(* IEC 61131-3 sources: eCockpitGit/test_project/src/%F%00 Library/%F%Common Functions/%F%Conversion/%F%AnyConversion, 28 files *)

(* ---- %POU%AnyATToSAny.st ---- *)
//This converts a pointer and a type to a sany
// |**Version**|**Author**| **Date** |**Changes**
// | 1         | NSN      | 13-12-19 | Creation
FUNCTION AnyATToSAny : SAny
VAR_INPUT
	pVal		:POINTER TO USysTypes;	//Address of value
	eType		:ESysType;				//Type of value
END_VAR
(*%!%__DELIMITER__%!%*)
AnyATToSAny.eType		:=		eType;
AnyATToSAny.pVal		:=		pVal;

(* ---- %POU%AnyToSAny.st ---- *)
//This function converts any variable to a sany
// |**Version**|**Author**| **Date** |**Changes**
// | 1         | NSN      | 13-12-19 | Creation
FUNCTION AnyToSAny : SAny
VAR_INPUT
	aAnyIn	:ANY;
END_VAR
(*%!%__DELIMITER__%!%*)
AnyToSAny.eType		:=		TO_BYTE(aAnyIn.TypeClass);
AnyToSAny.pVal		:=		aAnyIn.pValue;

(* ---- %POU%BitToSVar.st ---- *)
//This function get the bit value from a variable
// |**Version**|**Author**| **Date** |**Changes**
// | 1         | NSN      | 11-01-19 | Creation
FUNCTION BitToSVar : BOOL
VAR_INPUT
	xBit	:BOOL;		//Bool to set
	sVar	:SVar;		//Variable to get bit value from
END_VAR
(*%!%__DELIMITER__%!%*)
CASE sVar.bOffset OF
	1..8:	sVar.sAny.pVal^.bBYTE	:=		(sVar.sAny.pVal^.bBYTE AND NOT(SHL(TO_BYTE(1),sVar.bOffset-1))) OR (SHL(TO_BYTE(xBit),sVar.bOffset-1));
	9..16:	sVar.sAny.pVal^.bWORD	:=		(sVar.sAny.pVal^.bWORD AND NOT(SHL(TO_WORD(1),sVar.bOffset-1))) OR (SHL(TO_WORD(xBit),sVar.bOffset-1));
	17..32:	sVar.sAny.pVal^.bDWORD	:=		(sVar.sAny.pVal^.bDWORD AND NOT(SHL(TO_DWORD(1),sVar.bOffset-1))) OR (SHL(TO_DWORD(xBit),sVar.bOffset-1));
END_CASE

(* ---- %POU%BOOLToSAny.st ---- *)
//This function converts a dint to any variable
// |**Version**|**Author**| **Date** |**Changes**
// | 1         | NSN      | 23-07-18 | Creation
FUNCTION BOOLToSAny : BOOL
VAR_INPUT
	in			:BOOL;		//Input variable
	sOut		:SAny;		//Variable information
END_VAR
(*%!%__DELIMITER__%!%*)
CASE sOut.eType OF
	ESysType.tBOOL:		//Bool conversion
		sOut.pVal^.bBOOL		:=		in;
	ESysType.tBYTE:
		sOut.pVal^.bBYTE		:=		TO_BYTE(in);
	ESysType.tWORD:
		sOut.pVal^.bWORD		:=		TO_WORD(in);
	ESysType.tDWORD:
		sOut.pVal^.bDWORD		:=		TO_DWORD(in);
	ESysType.tLWORD:
		sOut.pVal^.bLWORD		:=		TO_LWORD(in);
	ESysType.tSINT:
		sOut.pVal^.bSINT		:=		TO_SINT(in);
	ESysType.tINT:
		sOut.pVal^.bINT			:=		TO_INT(in);
	ESysType.tDINT:
		sOut.pVal^.bDINT		:=		TO_DINT(in);
	ESysType.tLINT:
		sOut.pVal^.bLINT		:=		TO_LINT(in);
	ESysType.tUSINT:
		sOut.pVal^.bUSINT		:=		TO_USINT(in);
	ESysType.tUINT:
		sOut.pVal^.bUINT		:=		TO_UINT(in);
	ESysType.tUDINT:
		sOut.pVal^.bUDINT		:=		TO_UDINT(in);
	ESysType.tULINT:
		sOut.pVal^.bULINT		:=		TO_ULINT(in);
	ESysType.tREAL:
		sOut.pVal^.bREAL		:=		TO_REAL(in);
	ESysType.tLREAL:
		sOut.pVal^.bLREAL		:=		TO_LREAL(in);
	ESysType.tSTRING:
		sOut.pVal^.bSTRING		:=		TO_STRING(in);
	ESysType.tTIME:
		sOut.pVal^.bTIME		:=		TO_TIME(in);
	ESysType.tDATE:
		sOut.pVal^.bDATE		:=		TO_DATE(in);
	ESysType.tDT:
		sOut.pVal^.bDT			:=		TO_DT(in);
	ESysType.tTOD:
		sOut.pVal^.bTOD			:=		TO_TOD(in);
	ESysType.tLTIME:
		sOut.pVal^.bLTIME		:=		TO_LTIME(in);
ELSE
	RETURN;
END_CASE

(* ---- %POU%DINTToSAny.st ---- *)
//This function converts a dint to any variable
// |**Version**|**Author**| **Date** |**Changes**
// | 1         | NSN      | 23-07-18 | Creation
FUNCTION DINTToSAny : BOOL
VAR_INPUT
	in			:DINT;		//Input variable
	sOut		:SAny;		//Variable information
END_VAR
(*%!%__DELIMITER__%!%*)
CASE sOut.eType OF
	ESysType.tBOOL:		//Bool conversion
		sOut.pVal^.bBOOL		:=		TO_BOOL(in);
	ESysType.tBYTE:
		sOut.pVal^.bBYTE		:=		TO_BYTE(in);
	ESysType.tWORD:
		sOut.pVal^.bWORD		:=		TO_WORD(in);
	ESysType.tDWORD:
		sOut.pVal^.bDWORD		:=		TO_DWORD(in);
	ESysType.tLWORD:
		sOut.pVal^.bLWORD		:=		TO_LWORD(in);
	ESysType.tSINT:
		sOut.pVal^.bSINT		:=		TO_SINT(in);
	ESysType.tINT:
		sOut.pVal^.bINT			:=		TO_INT(in);
	ESysType.tDINT:
		sOut.pVal^.bDINT		:=		in;
	ESysType.tLINT:
		sOut.pVal^.bLINT		:=		in;
	ESysType.tUSINT:
		sOut.pVal^.bUSINT		:=		TO_USINT(in);
	ESysType.tUINT:
		sOut.pVal^.bUINT		:=		TO_UINT(in);
	ESysType.tUDINT:
		sOut.pVal^.bUDINT		:=		TO_UDINT(in);
	ESysType.tULINT:
		sOut.pVal^.bULINT		:=		TO_ULINT(in);
	ESysType.tREAL:
		sOut.pVal^.bREAL		:=		TO_REAL(in);
	ESysType.tLREAL:
		sOut.pVal^.bLREAL		:=		TO_LREAL(in);
	ESysType.tSTRING:
		sOut.pVal^.bSTRING		:=		TO_STRING(in);
	ESysType.tTIME:
		sOut.pVal^.bTIME		:=		TO_TIME(in);
	ESysType.tDATE:
		sOut.pVal^.bDATE		:=		TO_DATE(in);
	ESysType.tDT:
		sOut.pVal^.bDT			:=		TO_DT(in);
	ESysType.tTOD:
		sOut.pVal^.bTOD			:=		TO_TOD(in);
	ESysType.tLTIME:
		sOut.pVal^.bLTIME		:=		TO_LTIME(in);
ELSE
	RETURN;
END_CASE

(* ---- %POU%SAnyToBOOL.st ---- *)
//This function converts any type from the type and address to a real
// |**Version**|**Author**| **Date** |**Changes**
// | 1         | NSN      | 23-07-18 | Creation
FUNCTION SAnyToBOOL : BOOL
VAR_INPUT
	sAny		:SAny;		//Variable information
END_VAR
(*%!%__DELIMITER__%!%*)
CASE sAny.eType OF
	ESysType.tBOOL:		//Bool conversion
		SAnyToBOOL			:=		sAny.pVal^.bBOOL;
	ESysType.tBYTE:
		SAnyToBOOL			:=		TO_BOOL(sAny.pVal^.bBYTE);
	ESysType.tWORD:
		SAnyToBOOL			:=		TO_BOOL(sAny.pVal^.bWORD);
	ESysType.tDWORD:
		SAnyToBOOL			:=		TO_BOOL(sAny.pVal^.bDWORD);
	ESysType.tLWORD:
		SAnyToBOOL			:=		TO_BOOL(sAny.pVal^.bLWORD);
	ESysType.tSINT:
		SAnyToBOOL			:=		TO_BOOL(sAny.pVal^.bSINT);
	ESysType.tINT:
		SAnyToBOOL			:=		TO_BOOL(sAny.pVal^.bINT);
	ESysType.tDINT:
		SAnyToBOOL			:=		TO_BOOL(sAny.pVal^.bDINT);
	ESysType.tLINT:
		SAnyToBOOL			:=		TO_BOOL(sAny.pVal^.bLINT);
	ESysType.tUSINT:
		SAnyToBOOL			:=		TO_BOOL(sAny.pVal^.bUSINT);
	ESysType.tUINT:
		SAnyToBOOL			:=		TO_BOOL(sAny.pVal^.bUINT);
	ESysType.tUDINT:
		SAnyToBOOL			:=		TO_BOOL(sAny.pVal^.bUDINT);
	ESysType.tULINT:
		SAnyToBOOL			:=		TO_BOOL(sAny.pVal^.bULINT);
	ESysType.tREAL:
		SAnyToBOOL			:=		TO_BOOL(sAny.pVal^.bREAL);
	ESysType.tLREAL:
		SAnyToBOOL			:=		TO_BOOL(sAny.pVal^.bLREAL);
	ESysType.tSTRING:
		SAnyToBOOL			:=		TO_BOOL(sAny.pVal^.bSTRING);
	ESysType.tTIME:
		SAnyToBOOL			:=		TO_BOOL(sAny.pVal^.bTIME);
	ESysType.tDATE:
		SAnyToBOOL			:=		TO_BOOL(sAny.pVal^.bDATE);
	ESysType.tDT:
		SAnyToBOOL			:=		TO_BOOL(sAny.pVal^.bDT);
	ESysType.tTOD:
		SAnyToBOOL			:=		TO_BOOL(sAny.pVal^.bTOD);
	ESysType.tLTIME:
		SAnyToBOOL			:=		TO_BOOL(sAny.pVal^.bLTIME);
ELSE
	RETURN;
END_CASE

(* ---- %POU%SAnyToBYTE.st ---- *)
//This function converts any type from the type and address to a real
// |**Version**|**Author**| **Date** |**Changes**
// | 1         | NSN      | 23-07-18 | Creation
FUNCTION SAnyToBYTE : BYTE
VAR_INPUT
	sAny		:SAny;		//Variable information
END_VAR
(*%!%__DELIMITER__%!%*)
CASE sAny.eType OF
	ESysType.tBOOL:		//Bool conversion
		SAnyToBYTE			:=		TO_BYTE(sAny.pVal^.bBOOL);
	ESysType.tBYTE:
		SAnyToBYTE			:=		sAny.pVal^.bBYTE;
	ESysType.tWORD:
		SAnyToBYTE			:=		TO_BYTE(sAny.pVal^.bWORD);
	ESysType.tDWORD:
		SAnyToBYTE			:=		TO_BYTE(sAny.pVal^.bDWORD);
	ESysType.tLWORD:
		SAnyToBYTE			:=		TO_BYTE(sAny.pVal^.bLWORD);
	ESysType.tSINT:
		SAnyToBYTE			:=		TO_BYTE(sAny.pVal^.bSINT);
	ESysType.tINT:
		SAnyToBYTE			:=		TO_BYTE(sAny.pVal^.bINT);
	ESysType.tDINT:
		SAnyToBYTE			:=		TO_BYTE(sAny.pVal^.bDINT);
	ESysType.tLINT:
		SAnyToBYTE			:=		TO_BYTE(sAny.pVal^.bLINT);
	ESysType.tUSINT:
		SAnyToBYTE			:=		TO_BYTE(sAny.pVal^.bUSINT);
	ESysType.tUINT:
		SAnyToBYTE			:=		TO_BYTE(sAny.pVal^.bUINT);
	ESysType.tUDINT:
		SAnyToBYTE			:=		TO_BYTE(sAny.pVal^.bUDINT);
	ESysType.tULINT:
		SAnyToBYTE			:=		TO_BYTE(sAny.pVal^.bULINT);
	ESysType.tREAL:
		SAnyToBYTE			:=		TO_BYTE(sAny.pVal^.bREAL);
	ESysType.tLREAL:
		SAnyToBYTE			:=		TO_BYTE(sAny.pVal^.bLREAL);
	ESysType.tSTRING:
		SAnyToBYTE			:=		TO_BYTE(sAny.pVal^.bSTRING);
	ESysType.tTIME:
		SAnyToBYTE			:=		TO_BYTE(sAny.pVal^.bTIME);
	ESysType.tDATE:
		SAnyToBYTE			:=		TO_BYTE(sAny.pVal^.bDATE);
	ESysType.tDT:
		SAnyToBYTE			:=		TO_BYTE(sAny.pVal^.bDT);
	ESysType.tTOD:
		SAnyToBYTE			:=		TO_BYTE(sAny.pVal^.bTOD);
	ESysType.tLTIME:
		SAnyToBYTE			:=		TO_BYTE(sAny.pVal^.bLTIME);
ELSE
	RETURN;
END_CASE

(* ---- %POU%SAnyToDATE.st ---- *)
//This function converts any type from the type and address to a real
// |**Version**|**Author**| **Date** |**Changes**
// | 1         | NSN      | 23-07-18 | Creation
FUNCTION SAnyToDATE : DATE
VAR_INPUT
	sAny		:SAny;		//Variable information
END_VAR
(*%!%__DELIMITER__%!%*)
CASE sAny.eType OF
	ESysType.tBOOL:		//Bool conversion
		SAnyToDATE			:=		TO_DATE(sAny.pVal^.bBOOL);
	ESysType.tBYTE:
		SAnyToDATE			:=		TO_DATE(sAny.pVal^.bBYTE);
	ESysType.tWORD:
		SAnyToDATE			:=		TO_DATE(sAny.pVal^.bWORD);
	ESysType.tDWORD:
		SAnyToDATE			:=		TO_DATE(sAny.pVal^.bDWORD);
	ESysType.tLWORD:
		SAnyToDATE			:=		TO_DATE(sAny.pVal^.bLWORD);
	ESysType.tSINT:
		SAnyToDATE			:=		TO_DATE(sAny.pVal^.bSINT);
	ESysType.tINT:
		SAnyToDATE			:=		TO_DATE(sAny.pVal^.bINT);
	ESysType.tDINT:
		SAnyToDATE			:=		TO_DATE(sAny.pVal^.bDINT);
	ESysType.tLINT:
		SAnyToDATE			:=		TO_DATE(sAny.pVal^.bLINT);
	ESysType.tUSINT:
		SAnyToDATE			:=		TO_DATE(sAny.pVal^.bUSINT);
	ESysType.tUINT:
		SAnyToDATE			:=		TO_DATE(sAny.pVal^.bUINT);
	ESysType.tUDINT:
		SAnyToDATE			:=		TO_DATE(sAny.pVal^.bUDINT);
	ESysType.tULINT:
		SAnyToDATE			:=		TO_DATE(sAny.pVal^.bULINT);
	ESysType.tREAL:
		SAnyToDATE			:=		TO_DATE(sAny.pVal^.bREAL);
	ESysType.tLREAL:
		SAnyToDATE			:=		TO_DATE(sAny.pVal^.bLREAL);
	ESysType.tSTRING:
		SAnyToDATE			:=		TO_DATE(sAny.pVal^.bSTRING);
	ESysType.tTIME:
		SAnyToDATE			:=		TO_DATE(sAny.pVal^.bTIME);
	ESysType.tDATE:
		SAnyToDATE			:=		sAny.pVal^.bDATE;
	ESysType.tDT:
		SAnyToDATE			:=		TO_DATE(sAny.pVal^.bDT);
	ESysType.tTOD:
		SAnyToDATE			:=		TO_DATE(sAny.pVal^.bTOD);
	ESysType.tLTIME:
		SAnyToDATE			:=		TO_DATE(sAny.pVal^.bLTIME);
ELSE
	RETURN;
END_CASE

(* ---- %POU%SAnyToDINT.st ---- *)
//This function converts any type from the type and address to a real
// |**Version**|**Author**| **Date** |**Changes**
// | 1         | NSN      | 23-07-18 | Creation
FUNCTION SAnyToDINT : DINT
VAR_INPUT
	sAny		:SAny;		//Variable information
END_VAR
(*%!%__DELIMITER__%!%*)
CASE sAny.eType OF
	ESysType.tBOOL:		//Bool conversion
		SAnyToDINT			:=		TO_DINT(sAny.pVal^.bBOOL);
	ESysType.tBYTE:
		SAnyToDINT			:=		sAny.pVal^.bBYTE;
	ESysType.tWORD:
		SAnyToDINT			:=		sAny.pVal^.bWORD;
	ESysType.tDWORD:
		SAnyToDINT			:=		TO_DINT(sAny.pVal^.bDWORD);
	ESysType.tLWORD:
		SAnyToDINT			:=		TO_DINT(sAny.pVal^.bLWORD);
	ESysType.tSINT:
		SAnyToDINT			:=		sAny.pVal^.bSINT;
	ESysType.tINT:
		SAnyToDINT			:=		sAny.pVal^.bINT;
	ESysType.tDINT:
		SAnyToDINT			:=		sAny.pVal^.bDINT;
	ESysType.tLINT:
		SAnyToDINT			:=		TO_DINT(sAny.pVal^.bLINT);
	ESysType.tUSINT:
		SAnyToDINT			:=		sAny.pVal^.bUSINT;
	ESysType.tUINT:
		SAnyToDINT			:=		sAny.pVal^.bUINT;
	ESysType.tUDINT:
		SAnyToDINT			:=		TO_DINT(sAny.pVal^.bUDINT);
	ESysType.tULINT:
		SAnyToDINT			:=		TO_DINT(sAny.pVal^.bULINT);
	ESysType.tREAL:
		SAnyToDINT			:=		TO_DINT(sAny.pVal^.bREAL);
	ESysType.tLREAL:
		SAnyToDINT			:=		TO_DINT(sAny.pVal^.bLREAL);
	ESysType.tSTRING:
		SAnyToDINT			:=		TO_DINT(sAny.pVal^.bSTRING);
	ESysType.tTIME:
		SAnyToDINT			:=		TO_DINT(sAny.pVal^.bTIME);
	ESysType.tDATE:
		SAnyToDINT			:=		TO_DINT(sAny.pVal^.bDATE);
	ESysType.tDT:
		SAnyToDINT			:=		TO_DINT(sAny.pVal^.bDT);
	ESysType.tTOD:
		SAnyToDINT			:=		TO_DINT(sAny.pVal^.bTOD);
	ESysType.tLTIME:
		SAnyToDINT			:=		TO_DINT(sAny.pVal^.bLTIME);
ELSE
	RETURN;
END_CASE

(* ---- %POU%SAnyToDT.st ---- *)
//This function converts any type from the type and address to a real
// |**Version**|**Author**| **Date** |**Changes**
// | 1         | NSN      | 23-07-18 | Creation
FUNCTION SAnyToDT : DT
VAR_INPUT
	sAny		:SAny;		//Variable information
END_VAR
(*%!%__DELIMITER__%!%*)
CASE sAny.eType OF
	ESysType.tBOOL:		//Bool conversion
		SAnyToDT			:=		TO_DT(sAny.pVal^.bBOOL);
	ESysType.tBYTE:
		SAnyToDT			:=		TO_DT(sAny.pVal^.bBYTE);
	ESysType.tWORD:
		SAnyToDT			:=		TO_DT(sAny.pVal^.bWORD);
	ESysType.tDWORD:
		SAnyToDT			:=		TO_DT(sAny.pVal^.bDWORD);
	ESysType.tLWORD:
		SAnyToDT			:=		TO_DT(sAny.pVal^.bLWORD);
	ESysType.tSINT:
		SAnyToDT			:=		TO_DT(sAny.pVal^.bSINT);
	ESysType.tINT:
		SAnyToDT			:=		TO_DT(sAny.pVal^.bINT);
	ESysType.tDINT:
		SAnyToDT			:=		TO_DT(sAny.pVal^.bDINT);
	ESysType.tLINT:
		SAnyToDT			:=		TO_DT(sAny.pVal^.bLINT);
	ESysType.tUSINT:
		SAnyToDT			:=		TO_DT(sAny.pVal^.bUSINT);
	ESysType.tUINT:
		SAnyToDT			:=		TO_DT(sAny.pVal^.bUINT);
	ESysType.tUDINT:
		SAnyToDT			:=		TO_DT(sAny.pVal^.bUDINT);
	ESysType.tULINT:
		SAnyToDT			:=		TO_DT(sAny.pVal^.bULINT);
	ESysType.tREAL:
		SAnyToDT			:=		TO_DT(sAny.pVal^.bREAL);
	ESysType.tLREAL:
		SAnyToDT			:=		TO_DT(sAny.pVal^.bLREAL);
	ESysType.tSTRING:
		SAnyToDT			:=		TO_DT(sAny.pVal^.bSTRING);
	ESysType.tTIME:
		SAnyToDT			:=		TO_DT(sAny.pVal^.bTIME);
	ESysType.tDATE:
		SAnyToDT			:=		TO_DT(sAny.pVal^.bDATE);
	ESysType.tDT:
		SAnyToDT			:=		sAny.pVal^.bDT;
	ESysType.tTOD:
		SAnyToDT			:=		TO_DT(sAny.pVal^.bTOD);
	ESysType.tLTIME:
		SAnyToDT			:=		TO_DT(sAny.pVal^.bLTIME);
ELSE
	RETURN;
END_CASE

(* ---- %POU%SAnyToDWORD.st ---- *)
//This function converts any type from the type and address to a real
// |**Version**|**Author**| **Date** |**Changes**
// | 1         | NSN      | 23-07-18 | Creation
FUNCTION SAnyToDWORD : DWORD
VAR_INPUT
	sAny		:SAny;		//Variable information
END_VAR
(*%!%__DELIMITER__%!%*)
CASE sAny.eType OF
	ESysType.tBOOL:		//Bool conversion
		SAnyToDWORD			:=		TO_DWORD(sAny.pVal^.bBOOL);
	ESysType.tBYTE:
		SAnyToDWORD			:=		sAny.pVal^.bBYTE;
	ESysType.tWORD:
		SAnyToDWORD			:=		sAny.pVal^.bWORD;
	ESysType.tDWORD:
		SAnyToDWORD			:=		sAny.pVal^.bDWORD;
	ESysType.tLWORD:
		SAnyToDWORD			:=		TO_DWORD(sAny.pVal^.bLWORD);
	ESysType.tSINT:
		SAnyToDWORD			:=		TO_DWORD(sAny.pVal^.bSINT);
	ESysType.tINT:
		SAnyToDWORD			:=		TO_DWORD(sAny.pVal^.bINT);
	ESysType.tDINT:
		SAnyToDWORD			:=		TO_DWORD(sAny.pVal^.bDINT);
	ESysType.tLINT:
		SAnyToDWORD			:=		TO_DWORD(sAny.pVal^.bLINT);
	ESysType.tUSINT:
		SAnyToDWORD			:=		sAny.pVal^.bUSINT;
	ESysType.tUINT:
		SAnyToDWORD			:=		sAny.pVal^.bUINT;
	ESysType.tUDINT:
		SAnyToDWORD			:=		sAny.pVal^.bUDINT;
	ESysType.tULINT:
		SAnyToDWORD			:=		TO_DWORD(sAny.pVal^.bULINT);
	ESysType.tREAL:
		SAnyToDWORD			:=		TO_DWORD(sAny.pVal^.bREAL);
	ESysType.tLREAL:
		SAnyToDWORD			:=		TO_DWORD(sAny.pVal^.bLREAL);
	ESysType.tSTRING:
		SAnyToDWORD			:=		TO_DWORD(sAny.pVal^.bSTRING);
	ESysType.tTIME:
		SAnyToDWORD			:=		TO_DWORD(sAny.pVal^.bTIME);
	ESysType.tDATE:
		SAnyToDWORD			:=		TO_DWORD(sAny.pVal^.bDATE);
	ESysType.tDT:
		SAnyToDWORD			:=		TO_DWORD(sAny.pVal^.bDT);
	ESysType.tTOD:
		SAnyToDWORD			:=		TO_DWORD(sAny.pVal^.bTOD);
	ESysType.tLTIME:
		SAnyToDWORD			:=		TO_DWORD(sAny.pVal^.bLTIME);
ELSE
	RETURN;
END_CASE

(* ---- %POU%SAnyToINT.st ---- *)
//This function converts any type from the type and address to a real
// |**Version**|**Author**| **Date** |**Changes**
// | 1         | NSN      | 23-07-18 | Creation
FUNCTION SAnyToINT : INT
VAR_INPUT
	sAny		:SAny;		//Variable information
END_VAR
(*%!%__DELIMITER__%!%*)
CASE sAny.eType OF
	ESysType.tBOOL:		//Bool conversion
		SAnyToINT			:=		TO_INT(sAny.pVal^.bBOOL);
	ESysType.tBYTE:
		SAnyToINT			:=		sAny.pVal^.bBYTE;
	ESysType.tWORD:
		SAnyToINT			:=		TO_INT(sAny.pVal^.bWORD);
	ESysType.tDWORD:
		SAnyToINT			:=		TO_INT(sAny.pVal^.bDWORD);
	ESysType.tLWORD:
		SAnyToINT			:=		TO_INT(sAny.pVal^.bLWORD);
	ESysType.tSINT:
		SAnyToINT			:=		sAny.pVal^.bSINT;
	ESysType.tINT:
		SAnyToINT			:=		sAny.pVal^.bINT;
	ESysType.tDINT:
		SAnyToINT			:=		TO_INT(sAny.pVal^.bDINT);
	ESysType.tLINT:
		SAnyToINT			:=		TO_INT(sAny.pVal^.bLINT);
	ESysType.tUSINT:
		SAnyToINT			:=		sAny.pVal^.bUSINT;
	ESysType.tUINT:
		SAnyToINT			:=		TO_INT(sAny.pVal^.bUINT);
	ESysType.tUDINT:
		SAnyToINT			:=		TO_INT(sAny.pVal^.bUDINT);
	ESysType.tULINT:
		SAnyToINT			:=		TO_INT(sAny.pVal^.bULINT);
	ESysType.tREAL:
		SAnyToINT			:=		TO_INT(sAny.pVal^.bREAL);
	ESysType.tLREAL:
		SAnyToINT			:=		TO_INT(sAny.pVal^.bLREAL);
	ESysType.tSTRING:
		SAnyToINT			:=		TO_INT(sAny.pVal^.bSTRING);
	ESysType.tTIME:
		SAnyToINT			:=		TO_INT(sAny.pVal^.bTIME);
	ESysType.tDATE:
		SAnyToINT			:=		TO_INT(sAny.pVal^.bDATE);
	ESysType.tDT:
		SAnyToINT			:=		TO_INT(sAny.pVal^.bDT);
	ESysType.tTOD:
		SAnyToINT			:=		TO_INT(sAny.pVal^.bTOD);
	ESysType.tLTIME:
		SAnyToINT			:=		TO_INT(sAny.pVal^.bLTIME);
ELSE
	RETURN;
END_CASE

(* ---- %POU%SAnyToLINT.st ---- *)
//This function converts any type from the type and address to a real
// |**Version**|**Author**| **Date** |**Changes**
// | 1         | NSN      | 23-07-18 | Creation
FUNCTION SAnyToLINT : LINT
VAR_INPUT
	sAny		:SAny;		//Variable information
END_VAR
(*%!%__DELIMITER__%!%*)
CASE sAny.eType OF
	ESysType.tBOOL:		//Bool conversion
		SAnyToLINT			:=		TO_LINT(sAny.pVal^.bBOOL);
	ESysType.tBYTE:
		SAnyToLINT			:=		sAny.pVal^.bBYTE;
	ESysType.tWORD:
		SAnyToLINT			:=		sAny.pVal^.bWORD;
	ESysType.tDWORD:
		SAnyToLINT			:=		sAny.pVal^.bDWORD;
	ESysType.tLWORD:
		SAnyToLINT			:=		TO_LINT(sAny.pVal^.bLWORD);
	ESysType.tSINT:
		SAnyToLINT			:=		sAny.pVal^.bSINT;
	ESysType.tINT:
		SAnyToLINT			:=		sAny.pVal^.bINT;
	ESysType.tDINT:
		SAnyToLINT			:=		sAny.pVal^.bDINT;
	ESysType.tLINT:
		SAnyToLINT			:=		sAny.pVal^.bLINT;
	ESysType.tUSINT:
		SAnyToLINT			:=		sAny.pVal^.bUSINT;
	ESysType.tUINT:
		SAnyToLINT			:=		sAny.pVal^.bUINT;
	ESysType.tUDINT:
		SAnyToLINT			:=		sAny.pVal^.bUDINT;
	ESysType.tULINT:
		SAnyToLINT			:=		TO_LINT(sAny.pVal^.bULINT);
	ESysType.tREAL:
		SAnyToLINT			:=		TO_LINT(sAny.pVal^.bREAL);
	ESysType.tLREAL:
		SAnyToLINT			:=		TO_LINT(sAny.pVal^.bLREAL);
	ESysType.tSTRING:
		SAnyToLINT			:=		TO_LINT(sAny.pVal^.bSTRING);
	ESysType.tTIME:
		SAnyToLINT			:=		TO_LINT(sAny.pVal^.bTIME);
	ESysType.tDATE:
		SAnyToLINT			:=		TO_LINT(sAny.pVal^.bDATE);
	ESysType.tDT:
		SAnyToLINT			:=		TO_LINT(sAny.pVal^.bDT);
	ESysType.tTOD:
		SAnyToLINT			:=		TO_LINT(sAny.pVal^.bTOD);
	ESysType.tLTIME:
		SAnyToLINT			:=		TO_LINT(sAny.pVal^.bLTIME);
ELSE
	RETURN;
END_CASE

(* ---- %POU%SAnyToLREAL.st ---- *)
//This function converts any type from the type and address to a real
// |**Version**|**Author**| **Date** |**Changes**
// | 1         | NSN      | 23-07-18 | Creation
FUNCTION SAnyToLREAL : LREAL
VAR_INPUT
	sAny		:SAny;		//Variable information
END_VAR
(*%!%__DELIMITER__%!%*)
CASE sAny.eType OF
	ESysType.tBOOL:		//Bool conversion
		SAnyToLREAL			:=		TO_LREAL(sAny.pVal^.bBOOL);
	ESysType.tBYTE:
		SAnyToLREAL			:=		TO_LREAL(sAny.pVal^.bBYTE);
	ESysType.tWORD:
		SAnyToLREAL			:=		TO_LREAL(sAny.pVal^.bWORD);
	ESysType.tDWORD:
		SAnyToLREAL			:=		TO_LREAL(sAny.pVal^.bDWORD);
	ESysType.tLWORD:
		SAnyToLREAL			:=		TO_LREAL(sAny.pVal^.bLWORD);
	ESysType.tSINT:
		SAnyToLREAL			:=		TO_LREAL(sAny.pVal^.bSINT);
	ESysType.tINT:
		SAnyToLREAL			:=		TO_LREAL(sAny.pVal^.bINT);
	ESysType.tDINT:
		SAnyToLREAL			:=		TO_LREAL(sAny.pVal^.bDINT);
	ESysType.tLINT:
		SAnyToLREAL			:=		TO_LREAL(sAny.pVal^.bLINT);
	ESysType.tUSINT:
		SAnyToLREAL			:=		TO_LREAL(sAny.pVal^.bUSINT);
	ESysType.tUINT:
		SAnyToLREAL			:=		TO_LREAL(sAny.pVal^.bUINT);
	ESysType.tUDINT:
		SAnyToLREAL			:=		TO_LREAL(sAny.pVal^.bUDINT);
	ESysType.tULINT:
		SAnyToLREAL			:=		TO_LREAL(sAny.pVal^.bULINT);
	ESysType.tREAL:
		SAnyToLREAL			:=		sAny.pVal^.bREAL;
	ESysType.tLREAL:
		SAnyToLREAL			:=		sAny.pVal^.bLREAL;
	ESysType.tSTRING:
		SAnyToLREAL			:=		TO_LREAL(sAny.pVal^.bSTRING);
	ESysType.tTIME:
		SAnyToLREAL			:=		TO_LREAL(sAny.pVal^.bTIME);
	ESysType.tDATE:
		SAnyToLREAL			:=		TO_LREAL(sAny.pVal^.bDATE);
	ESysType.tDT:
		SAnyToLREAL			:=		TO_LREAL(sAny.pVal^.bDT);
	ESysType.tTOD:
		SAnyToLREAL			:=		TO_LREAL(sAny.pVal^.bTOD);
	ESysType.tLTIME:
		SAnyToLREAL			:=		TO_LREAL(sAny.pVal^.bLTIME);
ELSE
	RETURN;
END_CASE

(* ---- %POU%SAnyToLTIME.st ---- *)
//This function converts any type from the type and address to a real
// |**Version**|**Author**| **Date** |**Changes**
// | 1         | NSN      | 23-07-18 | Creation
FUNCTION SAnyToLTIME : LTIME
VAR_INPUT
	sAny		:SAny;		//Variable information
END_VAR
(*%!%__DELIMITER__%!%*)
CASE sAny.eType OF
	ESysType.tBOOL:		//Bool conversion
		SAnyToLTIME			:=		TO_LTIME(sAny.pVal^.bBOOL);
	ESysType.tBYTE:
		SAnyToLTIME			:=		TO_LTIME(sAny.pVal^.bBYTE);
	ESysType.tWORD:
		SAnyToLTIME			:=		TO_LTIME(sAny.pVal^.bWORD);
	ESysType.tDWORD:
		SAnyToLTIME			:=		TO_LTIME(sAny.pVal^.bDWORD);
	ESysType.tLWORD:
		SAnyToLTIME			:=		TO_LTIME(sAny.pVal^.bLWORD);
	ESysType.tSINT:
		SAnyToLTIME			:=		TO_LTIME(sAny.pVal^.bSINT);
	ESysType.tINT:
		SAnyToLTIME			:=		TO_LTIME(sAny.pVal^.bINT);
	ESysType.tDINT:
		SAnyToLTIME			:=		TO_LTIME(sAny.pVal^.bDINT);
	ESysType.tLINT:
		SAnyToLTIME			:=		TO_LTIME(sAny.pVal^.bLINT);
	ESysType.tUSINT:
		SAnyToLTIME			:=		TO_LTIME(sAny.pVal^.bUSINT);
	ESysType.tUINT:
		SAnyToLTIME			:=		TO_LTIME(sAny.pVal^.bUINT);
	ESysType.tUDINT:
		SAnyToLTIME			:=		TO_LTIME(sAny.pVal^.bUDINT);
	ESysType.tULINT:
		SAnyToLTIME			:=		TO_LTIME(sAny.pVal^.bULINT);
	ESysType.tREAL:
		SAnyToLTIME			:=		TO_LTIME(sAny.pVal^.bREAL);
	ESysType.tLREAL:
		SAnyToLTIME			:=		TO_LTIME(sAny.pVal^.bLREAL);
	ESysType.tSTRING:
		SAnyToLTIME			:=		TO_LTIME(sAny.pVal^.bSTRING);
	ESysType.tTIME:
		SAnyToLTIME			:=		TO_LTIME(sAny.pVal^.bTIME);
	ESysType.tDATE:
		SAnyToLTIME			:=		TO_LTIME(sAny.pVal^.bDATE);
	ESysType.tDT:
		SAnyToLTIME			:=		TO_LTIME(sAny.pVal^.bDT);
	ESysType.tTOD:
		SAnyToLTIME			:=		TO_LTIME(sAny.pVal^.bTOD);
	ESysType.tLTIME:
		SAnyToLTIME			:=		sAny.pVal^.bLTIME;
ELSE
	RETURN;
END_CASE

(* ---- %POU%SAnyToLWORD.st ---- *)
//This function converts any type from the type and address to a real
// |**Version**|**Author**| **Date** |**Changes**
// | 1         | NSN      | 23-07-18 | Creation
FUNCTION SAnyToLWORD : LWORD
VAR_INPUT
	sAny		:SAny;		//Variable information
END_VAR
(*%!%__DELIMITER__%!%*)
CASE sAny.eType OF
	ESysType.tBOOL:		//Bool conversion
		SAnyToLWORD			:=		TO_LWORD(sAny.pVal^.bBOOL);
	ESysType.tBYTE:
		SAnyToLWORD			:=		sAny.pVal^.bBYTE;
	ESysType.tWORD:
		SAnyToLWORD			:=		sAny.pVal^.bWORD;
	ESysType.tDWORD:
		SAnyToLWORD			:=		sAny.pVal^.bDWORD;
	ESysType.tLWORD:
		SAnyToLWORD			:=		sAny.pVal^.bLWORD;
	ESysType.tSINT:
		SAnyToLWORD			:=		TO_LWORD(sAny.pVal^.bSINT);
	ESysType.tINT:
		SAnyToLWORD			:=		TO_LWORD(sAny.pVal^.bINT);
	ESysType.tDINT:
		SAnyToLWORD			:=		TO_LWORD(sAny.pVal^.bDINT);
	ESysType.tLINT:
		SAnyToLWORD			:=		TO_LWORD(sAny.pVal^.bLINT);
	ESysType.tUSINT:
		SAnyToLWORD			:=		sAny.pVal^.bUSINT;
	ESysType.tUINT:
		SAnyToLWORD			:=		sAny.pVal^.bUINT;
	ESysType.tUDINT:
		SAnyToLWORD			:=		sAny.pVal^.bUDINT;
	ESysType.tULINT:
		SAnyToLWORD			:=		sAny.pVal^.bULINT;
	ESysType.tREAL:
		SAnyToLWORD			:=		TO_LWORD(sAny.pVal^.bREAL);
	ESysType.tLREAL:
		SAnyToLWORD			:=		TO_LWORD(sAny.pVal^.bLREAL);
	ESysType.tSTRING:
		SAnyToLWORD			:=		TO_LWORD(sAny.pVal^.bSTRING);
	ESysType.tTIME:
		SAnyToLWORD			:=		TO_LWORD(sAny.pVal^.bTIME);
	ESysType.tDATE:
		SAnyToLWORD			:=		TO_LWORD(sAny.pVal^.bDATE);
	ESysType.tDT:
		SAnyToLWORD			:=		TO_LWORD(sAny.pVal^.bDT);
	ESysType.tTOD:
		SAnyToLWORD			:=		TO_LWORD(sAny.pVal^.bTOD);
	ESysType.tLTIME:
		SAnyToLWORD			:=		TO_LWORD(sAny.pVal^.bLTIME);
ELSE
	RETURN;
END_CASE

(* ---- %POU%SAnyToREAL.st ---- *)
//This function converts any type from the type and address to a dint
// |**Version**|**Author**| **Date** |**Changes**
// | 1         | NSN      | 23-07-18 | Creation
FUNCTION SAnyToREAL : REAL
VAR_INPUT
	sAny		:SAny;		//Variable information
END_VAR
(*%!%__DELIMITER__%!%*)
CASE sAny.eType OF
	ESysType.tBOOL:		//Bool conversion
		SAnyToREAL			:=		TO_REAL(sAny.pVal^.bBOOL);
	ESysType.tBYTE:
		SAnyToREAL			:=		TO_REAL(sAny.pVal^.bBYTE);
	ESysType.tWORD:
		SAnyToREAL			:=		TO_REAL(sAny.pVal^.bWORD);
	ESysType.tDWORD:
		SAnyToREAL			:=		TO_REAL(sAny.pVal^.bDWORD);
	ESysType.tLWORD:
		SAnyToREAL			:=		TO_REAL(sAny.pVal^.bLWORD);
	ESysType.tSINT:
		SAnyToREAL			:=		TO_REAL(sAny.pVal^.bSINT);
	ESysType.tINT:
		SAnyToREAL			:=		TO_REAL(sAny.pVal^.bINT);
	ESysType.tDINT:
		SAnyToREAL			:=		TO_REAL(sAny.pVal^.bDINT);
	ESysType.tLINT:
		SAnyToREAL			:=		TO_REAL(sAny.pVal^.bLINT);
	ESysType.tUSINT:
		SAnyToREAL			:=		TO_REAL(sAny.pVal^.bUSINT);
	ESysType.tUINT:
		SAnyToREAL			:=		TO_REAL(sAny.pVal^.bUINT);
	ESysType.tUDINT:
		SAnyToREAL			:=		TO_REAL(sAny.pVal^.bUDINT);
	ESysType.tULINT:
		SAnyToREAL			:=		TO_REAL(sAny.pVal^.bULINT);
	ESysType.tREAL:
		SAnyToREAL			:=		sAny.pVal^.bREAL;
	ESysType.tLREAL:
		SAnyToREAL			:=		TO_REAL(sAny.pVal^.bLREAL);
	ESysType.tSTRING:
		SAnyToREAL			:=		TO_REAL(sAny.pVal^.bSTRING);
	ESysType.tTIME:
		SAnyToREAL			:=		TO_REAL(sAny.pVal^.bTIME);
	ESysType.tDATE:
		SAnyToREAL			:=		TO_REAL(sAny.pVal^.bDATE);
	ESysType.tDT:
		SAnyToREAL			:=		TO_REAL(sAny.pVal^.bDT);
	ESysType.tTOD:
		SAnyToREAL			:=		TO_REAL(sAny.pVal^.bTOD);
	ESysType.tLTIME:
		SAnyToREAL			:=		TO_REAL(sAny.pVal^.bLTIME);
ELSE
	RETURN;
END_CASE

(* ---- %POU%SAnyToSAny.st ---- *)
//This function converts any type from the type and address to any type
// |**Version**|**Author**| **Date** |**Changes**
// | 1         | NSN      | 07-12-18 | Creation
FUNCTION SAnyToSAny : BOOL
VAR_INPUT
	sAnyIn	:SAny;
	sAnyOut	:SAny;
END_VAR
(*%!%__DELIMITER__%!%*)
CASE sAnyOut.eType OF
	ESysType.tBOOL:		//Bool conversion
		sAnyOut.pVal^.bBOOL		:=		SAnyToBOOL(sAny:=sAnyIn);
	ESysType.tBYTE:
		sAnyOut.pVal^.bBYTE		:=		SAnyToBYTE(sAny:=sAnyIn);
	ESysType.tWORD:
		sAnyOut.pVal^.bWORD		:=		SAnyToWORD(sAny:=sAnyIn);
	ESysType.tDWORD:
		sAnyOut.pVal^.bDWORD	:=		SAnyToDWORD(sAny:=sAnyIn);
	ESysType.tLWORD:
		sAnyOut.pVal^.bLWORD	:=		SAnyToLWORD(sAny:=sAnyIn);
	ESysType.tSINT:
		sAnyOut.pVal^.bSINT		:=		SAnyToSINT(sAny:=sAnyIn);
	ESysType.tINT:
		sAnyOut.pVal^.bINT		:=		SAnyToINT(sAny:=sAnyIn);
	ESysType.tDINT:
		sAnyOut.pVal^.bDINT		:=		SAnyToDINT(sAny:=sAnyIn);
	ESysType.tLINT:
		sAnyOut.pVal^.bLINT		:=		SAnyToLINT(sAny:=sAnyIn);
	ESysType.tUSINT:
		sAnyOut.pVal^.bUSINT	:=		SAnyToUSINT(sAny:=sAnyIn);
	ESysType.tUINT:
		sAnyOut.pVal^.bUINT		:=		SAnyToUINT(sAny:=sAnyIn);
	ESysType.tUDINT:
		sAnyOut.pVal^.bUDINT	:=		SAnyToUDINT(sAny:=sAnyIn);
	ESysType.tULINT:
		sAnyOut.pVal^.bULINT	:=		SAnyToULINT(sAny:=sAnyIn);
	ESysType.tREAL:
		sAnyOut.pVal^.bREAL		:=		SAnyToREAL(sAny:=sAnyIn);
	ESysType.tLREAL:
		sAnyOut.pVal^.bLREAL	:=		SAnyToLREAL(sAny:=sAnyIn);
	ESysType.tSTRING:
		sAnyOut.pVal^.bSTRING	:=		SAnyToSTRING(sAny:=sAnyIn);
	ESysType.tTIME:
		sAnyOut.pVal^.bTIME		:=		SAnyToTIME(sAny:=sAnyIn);
	ESysType.tDATE:
		sAnyOut.pVal^.bDATE		:=		SAnyToDATE(sAny:=sAnyIn);
	ESysType.tDT:
		sAnyOut.pVal^.bDT		:=		SAnyToDT(sAny:=sAnyIn);
	ESysType.tTOD:
		sAnyOut.pVal^.bTOD		:=		SAnyToTOD(sAny:=sAnyIn);
	ESysType.tLTIME:
		sAnyOut.pVal^.bLTIME	:=		SAnyToLTIME(sAny:=sAnyIn);
ELSE
	SAnyToSAny					:=		TRUE;
	RETURN;
END_CASE

(* ---- %POU%SAnyToSINT.st ---- *)
//This function converts any type from the type and address to a real
// |**Version**|**Author**| **Date** |**Changes**
// | 1         | NSN      | 23-07-18 | Creation
FUNCTION SAnyToSINT : SINT
VAR_INPUT
	sAny		:SAny;		//Variable information
END_VAR
(*%!%__DELIMITER__%!%*)
CASE sAny.eType OF
	ESysType.tBOOL:		//Bool conversion
		SAnyToSINT			:=		TO_SINT(sAny.pVal^.bBOOL);
	ESysType.tBYTE:
		SAnyToSINT			:=		TO_SINT(sAny.pVal^.bBYTE);
	ESysType.tWORD:
		SAnyToSINT			:=		TO_SINT(sAny.pVal^.bWORD);
	ESysType.tDWORD:
		SAnyToSINT			:=		TO_SINT(sAny.pVal^.bDWORD);
	ESysType.tLWORD:
		SAnyToSINT			:=		TO_SINT(sAny.pVal^.bLWORD);
	ESysType.tSINT:
		SAnyToSINT			:=		sAny.pVal^.bSINT;
	ESysType.tINT:
		SAnyToSINT			:=		TO_SINT(sAny.pVal^.bINT);
	ESysType.tDINT:
		SAnyToSINT			:=		TO_SINT(sAny.pVal^.bDINT);
	ESysType.tLINT:
		SAnyToSINT			:=		TO_SINT(sAny.pVal^.bLINT);
	ESysType.tUSINT:
		SAnyToSINT			:=		TO_SINT(sAny.pVal^.bUSINT);
	ESysType.tUINT:
		SAnyToSINT			:=		TO_SINT(sAny.pVal^.bUINT);
	ESysType.tUDINT:
		SAnyToSINT			:=		TO_SINT(sAny.pVal^.bUDINT);
	ESysType.tULINT:
		SAnyToSINT			:=		TO_SINT(sAny.pVal^.bULINT);
	ESysType.tREAL:
		SAnyToSINT			:=		TO_SINT(sAny.pVal^.bREAL);
	ESysType.tLREAL:
		SAnyToSINT			:=		TO_SINT(sAny.pVal^.bLREAL);
	ESysType.tSTRING:
		SAnyToSINT			:=		TO_SINT(sAny.pVal^.bSTRING);
	ESysType.tTIME:
		SAnyToSINT			:=		TO_SINT(sAny.pVal^.bTIME);
	ESysType.tDATE:
		SAnyToSINT			:=		TO_SINT(sAny.pVal^.bDATE);
	ESysType.tDT:
		SAnyToSINT			:=		TO_SINT(sAny.pVal^.bDT);
	ESysType.tTOD:
		SAnyToSINT			:=		TO_SINT(sAny.pVal^.bTOD);
	ESysType.tLTIME:
		SAnyToSINT			:=		TO_SINT(sAny.pVal^.bLTIME);
ELSE
	RETURN;
END_CASE

(* ---- %POU%SAnyToSTRING.st ---- *)
//This function converts any type from the type and address to a real
// |**Version**|**Author**| **Date** |**Changes**
// | 1         | NSN      | 23-07-18 | Creation
FUNCTION SAnyToSTRING : STRING(80);
VAR_INPUT
	sAny		:SAny;		//Variable information
END_VAR
(*%!%__DELIMITER__%!%*)
CASE sAny.eType OF
	ESysType.tBOOL:		//Bool conversion
		SAnyToSTRING			:=		TO_STRING(sAny.pVal^.bBOOL);
	ESysType.tBYTE:
		SAnyToSTRING			:=		TO_STRING(sAny.pVal^.bBYTE);
	ESysType.tWORD:
		SAnyToSTRING			:=		TO_STRING(sAny.pVal^.bWORD);
	ESysType.tDWORD:
		SAnyToSTRING			:=		TO_STRING(sAny.pVal^.bDWORD);
	ESysType.tLWORD:
		SAnyToSTRING			:=		TO_STRING(sAny.pVal^.bLWORD);
	ESysType.tSINT:
		SAnyToSTRING			:=		TO_STRING(sAny.pVal^.bSINT);
	ESysType.tINT:
		SAnyToSTRING			:=		TO_STRING(sAny.pVal^.bINT);
	ESysType.tDINT:
		SAnyToSTRING			:=		TO_STRING(sAny.pVal^.bDINT);
	ESysType.tLINT:
		SAnyToSTRING			:=		TO_STRING(sAny.pVal^.bLINT);
	ESysType.tUSINT:
		SAnyToSTRING			:=		TO_STRING(sAny.pVal^.bUSINT);
	ESysType.tUINT:
		SAnyToSTRING			:=		TO_STRING(sAny.pVal^.bUINT);
	ESysType.tUDINT:
		SAnyToSTRING			:=		TO_STRING(sAny.pVal^.bUDINT);
	ESysType.tULINT:
		SAnyToSTRING			:=		TO_STRING(sAny.pVal^.bULINT);
	ESysType.tREAL:
		SAnyToSTRING			:=		TO_STRING(sAny.pVal^.bREAL);
	ESysType.tLREAL:
		SAnyToSTRING			:=		TO_STRING(sAny.pVal^.bLREAL);
	ESysType.tSTRING:
		SAnyToSTRING			:=		sAny.pVal^.bSTRING;
	ESysType.tTIME:
		SAnyToSTRING			:=		TO_STRING(sAny.pVal^.bTIME);
	ESysType.tDATE:
		SAnyToSTRING			:=		TO_STRING(sAny.pVal^.bDATE);
	ESysType.tDT:
		SAnyToSTRING			:=		TO_STRING(sAny.pVal^.bDT);
	ESysType.tTOD:
		SAnyToSTRING			:=		TO_STRING(sAny.pVal^.bTOD);
	ESysType.tLTIME:
		SAnyToSTRING			:=		TO_STRING(sAny.pVal^.bLTIME);
ELSE
	RETURN;
END_CASE

(* ---- %POU%SAnyToTIME.st ---- *)
//This function converts any type from the type and address to a real
// |**Version**|**Author**| **Date** |**Changes**
// | 1         | NSN      | 23-07-18 | Creation
FUNCTION SAnyToTIME : TIME
VAR_INPUT
	sAny		:SAny;		//Variable information
END_VAR
(*%!%__DELIMITER__%!%*)
CASE sAny.eType OF
	ESysType.tBOOL:		//Bool conversion
		SAnyToTIME			:=		TO_TIME(sAny.pVal^.bBOOL);
	ESysType.tBYTE:
		SAnyToTIME			:=		TO_TIME(sAny.pVal^.bBYTE);
	ESysType.tWORD:
		SAnyToTIME			:=		TO_TIME(sAny.pVal^.bWORD);
	ESysType.tDWORD:
		SAnyToTIME			:=		TO_TIME(sAny.pVal^.bDWORD);
	ESysType.tLWORD:
		SAnyToTIME			:=		TO_TIME(sAny.pVal^.bLWORD);
	ESysType.tSINT:
		SAnyToTIME			:=		TO_TIME(sAny.pVal^.bSINT);
	ESysType.tINT:
		SAnyToTIME			:=		TO_TIME(sAny.pVal^.bINT);
	ESysType.tDINT:
		SAnyToTIME			:=		TO_TIME(sAny.pVal^.bDINT);
	ESysType.tLINT:
		SAnyToTIME			:=		TO_TIME(sAny.pVal^.bLINT);
	ESysType.tUSINT:
		SAnyToTIME			:=		TO_TIME(sAny.pVal^.bUSINT);
	ESysType.tUINT:
		SAnyToTIME			:=		TO_TIME(sAny.pVal^.bUINT);
	ESysType.tUDINT:
		SAnyToTIME			:=		TO_TIME(sAny.pVal^.bUDINT);
	ESysType.tULINT:
		SAnyToTIME			:=		TO_TIME(sAny.pVal^.bULINT);
	ESysType.tREAL:
		SAnyToTIME			:=		TO_TIME(sAny.pVal^.bREAL);
	ESysType.tLREAL:
		SAnyToTIME			:=		TO_TIME(sAny.pVal^.bLREAL);
	ESysType.tSTRING:
		SAnyToTIME			:=		TO_TIME(sAny.pVal^.bSTRING);
	ESysType.tTIME:
		SAnyToTIME			:=		sAny.pVal^.bTIME;
	ESysType.tDATE:
		SAnyToTIME			:=		TO_TIME(sAny.pVal^.bDATE);
	ESysType.tDT:
		SAnyToTIME			:=		TO_TIME(sAny.pVal^.bDT);
	ESysType.tTOD:
		SAnyToTIME			:=		TO_TIME(sAny.pVal^.bTOD);
	ESysType.tLTIME:
		SAnyToTIME			:=		TO_TIME(sAny.pVal^.bLTIME);
ELSE
	RETURN;
END_CASE

(* ---- %POU%SAnyToTOD.st ---- *)
//This function converts any type from the type and address to a real
// |**Version**|**Author**| **Date** |**Changes**
// | 1         | NSN      | 23-07-18 | Creation
FUNCTION SAnyToTOD : TOD
VAR_INPUT
	sAny		:SAny;		//Variable information
END_VAR
(*%!%__DELIMITER__%!%*)
CASE sAny.eType OF
	ESysType.tBOOL:		//Bool conversion
		SAnyToTOD			:=		TO_TOD(sAny.pVal^.bBOOL);
	ESysType.tBYTE:
		SAnyToTOD			:=		TO_TOD(sAny.pVal^.bBYTE);
	ESysType.tWORD:
		SAnyToTOD			:=		TO_TOD(sAny.pVal^.bWORD);
	ESysType.tDWORD:
		SAnyToTOD			:=		TO_TOD(sAny.pVal^.bDWORD);
	ESysType.tLWORD:
		SAnyToTOD			:=		TO_TOD(sAny.pVal^.bLWORD);
	ESysType.tSINT:
		SAnyToTOD			:=		TO_TOD(sAny.pVal^.bSINT);
	ESysType.tINT:
		SAnyToTOD			:=		TO_TOD(sAny.pVal^.bINT);
	ESysType.tDINT:
		SAnyToTOD			:=		TO_TOD(sAny.pVal^.bDINT);
	ESysType.tLINT:
		SAnyToTOD			:=		TO_TOD(sAny.pVal^.bLINT);
	ESysType.tUSINT:
		SAnyToTOD			:=		TO_TOD(sAny.pVal^.bUSINT);
	ESysType.tUINT:
		SAnyToTOD			:=		TO_TOD(sAny.pVal^.bUINT);
	ESysType.tUDINT:
		SAnyToTOD			:=		TO_TOD(sAny.pVal^.bUDINT);
	ESysType.tULINT:
		SAnyToTOD			:=		TO_TOD(sAny.pVal^.bULINT);
	ESysType.tREAL:
		SAnyToTOD			:=		TO_TOD(sAny.pVal^.bREAL);
	ESysType.tLREAL:
		SAnyToTOD			:=		TO_TOD(sAny.pVal^.bLREAL);
	ESysType.tSTRING:
		SAnyToTOD			:=		TO_TOD(sAny.pVal^.bSTRING);
	ESysType.tTIME:
		SAnyToTOD			:=		TO_TOD(sAny.pVal^.bTIME);
	ESysType.tDATE:
		SAnyToTOD			:=		TO_TOD(sAny.pVal^.bDATE);
	ESysType.tDT:
		SAnyToTOD			:=		TO_TOD(sAny.pVal^.bDT);
	ESysType.tTOD:
		SAnyToTOD			:=		sAny.pVal^.bTOD;
	ESysType.tLTIME:
		SAnyToTOD			:=		TO_TOD(sAny.pVal^.bLTIME);
ELSE
	RETURN;
END_CASE

(* ---- %POU%SAnyToUDINT.st ---- *)
//This function converts any type from the type and address to a real
// |**Version**|**Author**| **Date** |**Changes**
// | 1         | NSN      | 23-07-18 | Creation
FUNCTION SAnyToUDINT : UDINT
VAR_INPUT
	sAny		:SAny;		//Variable information
END_VAR
(*%!%__DELIMITER__%!%*)
CASE sAny.eType OF
	ESysType.tBOOL:		//Bool conversion
		SAnyToUDINT			:=		TO_UDINT(sAny.pVal^.bBOOL);
	ESysType.tBYTE:
		SAnyToUDINT			:=		sAny.pVal^.bBYTE;
	ESysType.tWORD:
		SAnyToUDINT			:=		sAny.pVal^.bWORD;
	ESysType.tDWORD:
		SAnyToUDINT			:=		sAny.pVal^.bDWORD;
	ESysType.tLWORD:
		SAnyToUDINT			:=		TO_UDINT(sAny.pVal^.bLWORD);
	ESysType.tSINT:
		SAnyToUDINT			:=		TO_UDINT(sAny.pVal^.bSINT);
	ESysType.tINT:
		SAnyToUDINT			:=		TO_UDINT(sAny.pVal^.bINT);
	ESysType.tDINT:
		SAnyToUDINT			:=		TO_UDINT(sAny.pVal^.bDINT);
	ESysType.tLINT:
		SAnyToUDINT			:=		TO_UDINT(sAny.pVal^.bLINT);
	ESysType.tUSINT:
		SAnyToUDINT			:=		sAny.pVal^.bUSINT;
	ESysType.tUINT:
		SAnyToUDINT			:=		sAny.pVal^.bUINT;
	ESysType.tUDINT:
		SAnyToUDINT			:=		sAny.pVal^.bUDINT;
	ESysType.tULINT:
		SAnyToUDINT			:=		TO_UDINT(sAny.pVal^.bULINT);
	ESysType.tREAL:
		SAnyToUDINT			:=		TO_UDINT(sAny.pVal^.bREAL);
	ESysType.tLREAL:
		SAnyToUDINT			:=		TO_UDINT(sAny.pVal^.bLREAL);
	ESysType.tSTRING:
		SAnyToUDINT			:=		TO_UDINT(sAny.pVal^.bSTRING);
	ESysType.tTIME:
		SAnyToUDINT			:=		TO_UDINT(sAny.pVal^.bTIME);
	ESysType.tDATE:
		SAnyToUDINT			:=		TO_UDINT(sAny.pVal^.bDATE);
	ESysType.tDT:
		SAnyToUDINT			:=		TO_UDINT(sAny.pVal^.bDT);
	ESysType.tTOD:
		SAnyToUDINT			:=		TO_UDINT(sAny.pVal^.bTOD);
	ESysType.tLTIME:
		SAnyToUDINT			:=		TO_UDINT(sAny.pVal^.bLTIME);
ELSE
	RETURN;
END_CASE

(* ---- %POU%SAnyToUINT.st ---- *)
//This function converts any type from the type and address to a real
// |**Version**|**Author**| **Date** |**Changes**
// | 1         | NSN      | 23-07-18 | Creation
FUNCTION SAnyToUINT : UINT
VAR_INPUT
	sAny		:SAny;		//Variable information
END_VAR
(*%!%__DELIMITER__%!%*)
CASE sAny.eType OF
	ESysType.tBOOL:		//Bool conversion
		SAnyToUINT			:=		TO_UINT(sAny.pVal^.bBOOL);
	ESysType.tBYTE:
		SAnyToUINT			:=		sAny.pVal^.bBYTE;
	ESysType.tWORD:
		SAnyToUINT			:=		sAny.pVal^.bWORD;
	ESysType.tDWORD:
		SAnyToUINT			:=		TO_UINT(sAny.pVal^.bDWORD);
	ESysType.tLWORD:
		SAnyToUINT			:=		TO_UINT(sAny.pVal^.bLWORD);
	ESysType.tSINT:
		SAnyToUINT			:=		TO_UINT(sAny.pVal^.bSINT);
	ESysType.tINT:
		SAnyToUINT			:=		TO_UINT(sAny.pVal^.bINT);
	ESysType.tDINT:
		SAnyToUINT			:=		TO_UINT(sAny.pVal^.bDINT);
	ESysType.tLINT:
		SAnyToUINT			:=		TO_UINT(sAny.pVal^.bLINT);
	ESysType.tUSINT:
		SAnyToUINT			:=		sAny.pVal^.bUSINT;
	ESysType.tUINT:
		SAnyToUINT			:=		sAny.pVal^.bUINT;
	ESysType.tUDINT:
		SAnyToUINT			:=		TO_UINT(sAny.pVal^.bUDINT);
	ESysType.tULINT:
		SAnyToUINT			:=		TO_UINT(sAny.pVal^.bULINT);
	ESysType.tREAL:
		SAnyToUINT			:=		TO_UINT(sAny.pVal^.bREAL);
	ESysType.tLREAL:
		SAnyToUINT			:=		TO_UINT(sAny.pVal^.bLREAL);
	ESysType.tSTRING:
		SAnyToUINT			:=		TO_UINT(sAny.pVal^.bSTRING);
	ESysType.tTIME:
		SAnyToUINT			:=		TO_UINT(sAny.pVal^.bTIME);
	ESysType.tDATE:
		SAnyToUINT			:=		TO_UINT(sAny.pVal^.bDATE);
	ESysType.tDT:
		SAnyToUINT			:=		TO_UINT(sAny.pVal^.bDT);
	ESysType.tTOD:
		SAnyToUINT			:=		TO_UINT(sAny.pVal^.bTOD);
	ESysType.tLTIME:
		SAnyToUINT			:=		TO_UINT(sAny.pVal^.bLTIME);
ELSE
	RETURN;
END_CASE

(* ---- %POU%SAnyToULINT.st ---- *)
//This function converts any type from the type and address to a real
// |**Version**|**Author**| **Date** |**Changes**
// | 1         | NSN      | 23-07-18 | Creation
FUNCTION SAnyToULINT : ULINT
VAR_INPUT
	sAny		:SAny;		//Variable information
END_VAR
(*%!%__DELIMITER__%!%*)
CASE sAny.eType OF
	ESysType.tBOOL:		//Bool conversion
		SAnyToULINT			:=		TO_ULINT(sAny.pVal^.bBOOL);
	ESysType.tBYTE:
		SAnyToULINT			:=		TO_ULINT(sAny.pVal^.bBYTE);
	ESysType.tWORD:
		SAnyToULINT			:=		TO_ULINT(sAny.pVal^.bWORD);
	ESysType.tDWORD:
		SAnyToULINT			:=		TO_ULINT(sAny.pVal^.bDWORD);
	ESysType.tLWORD:
		SAnyToULINT			:=		TO_ULINT(sAny.pVal^.bLWORD);
	ESysType.tSINT:
		SAnyToULINT			:=		TO_ULINT(sAny.pVal^.bSINT);
	ESysType.tINT:
		SAnyToULINT			:=		TO_ULINT(sAny.pVal^.bINT);
	ESysType.tDINT:
		SAnyToULINT			:=		TO_ULINT(sAny.pVal^.bDINT);
	ESysType.tLINT:
		SAnyToULINT			:=		TO_ULINT(sAny.pVal^.bLINT);
	ESysType.tUSINT:
		SAnyToULINT			:=		TO_ULINT(sAny.pVal^.bUSINT);
	ESysType.tUINT:
		SAnyToULINT			:=		TO_ULINT(sAny.pVal^.bUINT);
	ESysType.tUDINT:
		SAnyToULINT			:=		TO_ULINT(sAny.pVal^.bUDINT);
	ESysType.tULINT:
		SAnyToULINT			:=		TO_ULINT(sAny.pVal^.bULINT);
	ESysType.tREAL:
		SAnyToULINT			:=		TO_ULINT(sAny.pVal^.bREAL);
	ESysType.tLREAL:
		SAnyToULINT			:=		TO_ULINT(sAny.pVal^.bLREAL);
	ESysType.tSTRING:
		SAnyToULINT			:=		TO_ULINT(sAny.pVal^.bSTRING);
	ESysType.tTIME:
		SAnyToULINT			:=		TO_ULINT(sAny.pVal^.bTIME);
	ESysType.tDATE:
		SAnyToULINT			:=		TO_ULINT(sAny.pVal^.bDATE);
	ESysType.tDT:
		SAnyToULINT			:=		TO_ULINT(sAny.pVal^.bDT);
	ESysType.tTOD:
		SAnyToULINT			:=		TO_ULINT(sAny.pVal^.bTOD);
	ESysType.tLTIME:
		SAnyToULINT			:=		TO_ULINT(sAny.pVal^.bLTIME);
ELSE
	RETURN;
END_CASE

(* ---- %POU%SAnyToUSINT.st ---- *)
//This function converts any type from the type and address to a real
// |**Version**|**Author**| **Date** |**Changes**
// | 1         | NSN      | 23-07-18 | Creation
FUNCTION SAnyToUSINT : USINT
VAR_INPUT
	sAny		:SAny;		//Variable information
END_VAR
(*%!%__DELIMITER__%!%*)
CASE sAny.eType OF
	ESysType.tBOOL:
		SAnyToUSINT			:=		TO_USINT(sAny.pVal^.bBOOL);
	ESysType.tBYTE:
		SAnyToUSINT			:=		sAny.pVal^.bBYTE;
	ESysType.tWORD:
		SAnyToUSINT			:=		TO_USINT(sAny.pVal^.bWORD);
	ESysType.tDWORD:
		SAnyToUSINT			:=		TO_USINT(sAny.pVal^.bDWORD);
	ESysType.tLWORD:
		SAnyToUSINT			:=		TO_USINT(sAny.pVal^.bLWORD);
	ESysType.tSINT:
		SAnyToUSINT			:=		TO_USINT(sAny.pVal^.bSINT);
	ESysType.tINT:
		SAnyToUSINT			:=		TO_USINT(sAny.pVal^.bINT);
	ESysType.tDINT:
		SAnyToUSINT			:=		TO_USINT(sAny.pVal^.bDINT);
	ESysType.tLINT:
		SAnyToUSINT			:=		TO_USINT(sAny.pVal^.bLINT);
	ESysType.tUSINT:
		SAnyToUSINT			:=		sAny.pVal^.bUSINT;
	ESysType.tUINT:
		SAnyToUSINT			:=		TO_USINT(sAny.pVal^.bUINT);
	ESysType.tUDINT:
		SAnyToUSINT			:=		TO_USINT(sAny.pVal^.bUDINT);
	ESysType.tULINT:
		SAnyToUSINT			:=		TO_USINT(sAny.pVal^.bULINT);
	ESysType.tREAL:
		SAnyToUSINT			:=		TO_USINT(sAny.pVal^.bREAL);
	ESysType.tLREAL:
		SAnyToUSINT			:=		TO_USINT(sAny.pVal^.bLREAL);
	ESysType.tSTRING:
		SAnyToUSINT			:=		TO_USINT(sAny.pVal^.bSTRING);
	ESysType.tTIME:
		SAnyToUSINT			:=		TO_USINT(sAny.pVal^.bTIME);
	ESysType.tDATE:
		SAnyToUSINT			:=		TO_USINT(sAny.pVal^.bDATE);
	ESysType.tDT:
		SAnyToUSINT			:=		TO_USINT(sAny.pVal^.bDT);
	ESysType.tTOD:
		SAnyToUSINT			:=		TO_USINT(sAny.pVal^.bTOD);
	ESysType.tLTIME:
		SAnyToUSINT			:=		TO_USINT(sAny.pVal^.bLTIME);
ELSE
	RETURN;
END_CASE

(* ---- %POU%SAnyToWORD.st ---- *)
//This function converts any type from the type and address to a real
// |**Version**|**Author**| **Date** |**Changes**
// | 1         | NSN      | 23-07-18 | Creation
FUNCTION SAnyToWORD : WORD
VAR_INPUT
	sAny		:SAny;		//Variable information
END_VAR
(*%!%__DELIMITER__%!%*)
CASE sAny.eType OF
	ESysType.tBOOL:		//Bool conversion
		SAnyToWORD			:=		TO_WORD(sAny.pVal^.bBOOL);
	ESysType.tBYTE:
		SAnyToWORD			:=		sAny.pVal^.bBYTE;
	ESysType.tWORD:
		SAnyToWORD			:=		sAny.pVal^.bWORD;
	ESysType.tDWORD:
		SAnyToWORD			:=		TO_WORD(sAny.pVal^.bDWORD);
	ESysType.tLWORD:
		SAnyToWORD			:=		TO_WORD(sAny.pVal^.bLWORD);
	ESysType.tSINT:
		SAnyToWORD			:=		TO_WORD(sAny.pVal^.bSINT);
	ESysType.tINT:
		SAnyToWORD			:=		TO_WORD(sAny.pVal^.bINT);
	ESysType.tDINT:
		SAnyToWORD			:=		TO_WORD(sAny.pVal^.bDINT);
	ESysType.tLINT:
		SAnyToWORD			:=		TO_WORD(sAny.pVal^.bLINT);
	ESysType.tUSINT:
		SAnyToWORD			:=		sAny.pVal^.bUSINT;
	ESysType.tUINT:
		SAnyToWORD			:=		sAny.pVal^.bUINT;
	ESysType.tUDINT:
		SAnyToWORD			:=		TO_WORD(sAny.pVal^.bUDINT);
	ESysType.tULINT:
		SAnyToWORD			:=		TO_WORD(sAny.pVal^.bULINT);
	ESysType.tREAL:
		SAnyToWORD			:=		TO_WORD(sAny.pVal^.bREAL);
	ESysType.tLREAL:
		SAnyToWORD			:=		TO_WORD(sAny.pVal^.bLREAL);
	ESysType.tSTRING:
		SAnyToWORD			:=		TO_WORD(sAny.pVal^.bSTRING);
	ESysType.tTIME:
		SAnyToWORD			:=		TO_WORD(sAny.pVal^.bTIME);
	ESysType.tDATE:
		SAnyToWORD			:=		TO_WORD(sAny.pVal^.bDATE);
	ESysType.tDT:
		SAnyToWORD			:=		TO_WORD(sAny.pVal^.bDT);
	ESysType.tTOD:
		SAnyToWORD			:=		TO_WORD(sAny.pVal^.bTOD);
	ESysType.tLTIME:
		SAnyToWORD			:=		TO_WORD(sAny.pVal^.bLTIME);
ELSE
	RETURN;
END_CASE

(* ---- %POU%SVarToBit.st ---- *)
//This function get the bit value from a variable
// |**Version**|**Author**| **Date** |**Changes**
// | 1         | NSN      | 11-01-19 | Creation
FUNCTION SVarToBit : BOOL
VAR_INPUT
	sVar	:SVar;		//Variable to get bit value from
END_VAR
(*%!%__DELIMITER__%!%*)
CASE sVar.bOffset OF
	1..8:	SVarToBit		:=		(sVar.sAny.pVal^.bBYTE AND SHL(1,sVar.bOffset-1)) <> 0;
	9..16:	SVarToBit		:=		(sVar.sAny.pVal^.bWORD AND SHL(1,sVar.bOffset-1)) <> 0;
	17..32:	SVarToBit		:=		(sVar.sAny.pVal^.bDWORD AND SHL(1,sVar.bOffset-1)) <> 0;
END_CASE
